(* CODESYS project FU_rMinMaxValue.xml

Project tree, tasks and I/O mapping:
  function FU_rMinMaxValue [ST]
*)

// FU_rMinMaxValue
//This function keeps a variable between a minimum and a maximum value
// +-----------+----------+----------+-----------------------------------------------------------------------------------------------------------------------+
// |**Version**|**Author**| **Date** |**Changes**                                                                                                            |
// +-----------+----------+----------+-----------------------------------------------------------------------------------------------------------------------+
// | 1         | NSN      | 07-01-18 | Creation                                                                                                              |
// +-----------+----------+----------+-----------------------------------------------------------------------------------------------------------------------+
FUNCTION FU_rMinMaxValue : BOOL
VAR_IN_OUT
	Variable		:REAL;
END_VAR
VAR_INPUT
	MinVal			:REAL;
	MaxVal			:REAL;
END_VAR

IF Variable < MinVal THEN			//This makes sure only values between minval and maxval can be entered
	Variable				:=		MinVal;
ELSIF Variable > MaxVal THEN
	Variable				:=		MaxVal;
END_IF

END_FUNCTION
